FUNCTION_BLOCK FB_Bimanual EXTENDS FB_Device
VAR_INPUT
	diStationState					: EN_StationStatus;
END_VAR
VAR
	Sensor 				AT %I* 		: BOOL;	
	Green 				AT %Q* 		: BOOL;
	Ambar 				AT %Q* 		: BOOL;
	Red 				AT %Q* 		: BOOL;
	Blink 				AT %Q* 		: BOOL;
	END_VAR

END_FUNCTION_BLOCK

(* stored: Version 1.1.0.1
   POU FB_Bimanual: Id {a5709532-78d9-4de9-b90c-12c4dc9054e6}, SpecialFunc None *)
